			IF curStep = 1 THEN
				IF ZeitPuls > loc_ET_ms THEN
					RestzeitPuls := ZeitPuls - loc_ET_ms;
				ELSE
					RestzeitPuls := 0;
				END_IF;
				RestzeitPause := ZeitPause;
			ELSE
				RestzeitPuls := ZeitPuls;
				IF ZeitPause > loc_ET_ms THEN
					RestzeitPause := ZeitPause - loc_ET_ms;
				ELSE
					RestzeitPause := 0;
				END_IF;
			END_IF;
		END_IF;

	END_IF;

ELSE
	(* keine Freigabe -> Schrittkette ruecksetzen *)
	PulsOut       := FALSE;
	PauseOut      := FALSE;
	RestzeitPuls  := 0;
	RestzeitPause := 0;
	TON_PulsPause(IN := FALSE, PT := 0);
	curStep       := 0;
	stateEntry    := TRUE;
END_IF;
END_FUNCTION_BLOCK

FUNCTION_BLOCK fbRestzeit
  VAR
    i : INT;
    ii : INT;
    stundeEndeTag : INT;
    minRestTag : UINT;
    minRestFolgetag : UINT;
    minRestGesamt : UINT;
    restStd : UINT;
  END_VAR
  VAR_INPUT
    Freigabe : BOOL;
    AktuelleStunde : USINT;  (* 0..23 *)
    AktuelleMinute : USINT;  (* 0..59 *)
  END_VAR
  VAR_OUTPUT
    ZeitfensterAktiv : BOOL;
    RestzeitStundenOut : UINT;
    RestzeitMinutenOut : UINT;
  END_VAR
  VAR_IN_OUT
    ZeitfensterIn : ARRAY[0..23] OF BOOL;
  END_VAR

IF Freigabe THEN
    ZeitfensterAktiv := ZeitfensterIn[AktuelleStunde];

    (* Ende des aktuellen (gleichbleibenden) Blocks heute suchen *)
    stundeEndeTag := 23;
    FOR i := TO_INT(AktuelleStunde) + 1 TO 23 DO
        IF ZeitfensterIn[i] <> ZeitfensterAktiv THEN
            stundeEndeTag := i - 1;
            EXIT;
        END_IF;
    END_FOR;

    (* Restminuten heute *)
    minRestTag := 60 - AktuelleMinute;
    IF stundeEndeTag > TO_INT(AktuelleStunde) THEN
        minRestTag := minRestTag + TO_UINT(stundeEndeTag - TO_INT(AktuelleStunde)) * 60;
    END_IF;

    (* Folgetag nur, wenn Block bis 23 Uhr durchlaeuft *)
    minRestFolgetag := 0;
    IF stundeEndeTag = 23 THEN
        FOR ii := 0 TO 23 DO
            IF ZeitfensterIn[ii] = ZeitfensterAktiv THEN
                minRestFolgetag := minRestFolgetag + 60;
            ELSE
                EXIT;
            END_IF;
        END_FOR;
    END_IF;

    minRestGesamt := minRestTag + minRestFolgetag;
    restStd := minRestGesamt / 60;
    IF restStd <= 24 THEN
        RestzeitStundenOut := restStd;
        RestzeitMinutenOut := minRestGesamt - (restStd * 60);
    ELSE
        RestzeitStundenOut := 65535;   (* >24h -> keine Anzeige *)
        RestzeitMinutenOut := 65535;
    END_IF;
ELSE
    ZeitfensterAktiv   := FALSE;
    RestzeitStundenOut := 65535;
    RestzeitMinutenOut := 65535;
END_IF;
END_FUNCTION_BLOCK

FUNCTION_BLOCK fbBetriebsstunden
  VAR
    Sekunden : USINT;
  END_VAR
  VAR_INPUT
    Aktiv : BOOL;
    sekTick : BOOL;  (* 1-Sekunden-Puls *)
    Reset : BOOL;
  END_VAR
  VAR_IN_OUT
    Minuten : UINT;  (* Retain-Global, 0..59 *)
    Stunden : UDINT;  (* Retain-Global *)
  END_VAR

IF Reset THEN
    Sekunden := 0;  Minuten := 0;  Stunden := 0;
ELSIF (Aktiv AND sekTick) THEN
    IF Sekunden < 59 THEN
        Sekunden := Sekunden + 1;
    ELSE
        Sekunden := 0;
        IF Minuten < 59 THEN
            Minuten := Minuten + 1;
        ELSE
            Minuten := 0;
            Stunden := Stunden + 1;
        END_IF;
    END_IF;
END_IF;
END_FUNCTION_BLOCK

FUNCTION fcSetBitInBitmask : UDINT
  VAR
    ValBit : UDINT;
  END_VAR
  VAR_INPUT
    Bitmask : UDINT;
    BitNr : USINT;
  END_VAR

// Bitstelle in Wert umwandeln
ValBit := SHL(UDINT#1, BitNr);

// Bit in Bitmaske setzen
fcSetBitInBitmask := Bitmask OR ValBit;
END_FUNCTION

FUNCTION fcClearBitInBitmask : UDINT
  VAR
    ValBit : UDINT;
  END_VAR
  VAR_INPUT
    Bitmask : UDINT;
    BitNr : USINT;
  END_VAR

// Bitstelle in Wert umwandeln
ValBit := SHL(UDINT#1, BitNr);

// Bit in Bitmaske löschen
fcClearBitInBitmask := Bitmask AND NOT ValBit;
END_FUNCTION

FUNCTION fcResetBitmask : UDINT

fcResetBitmask := TO_UDINT(0);
END_FUNCTION

CONFIGURATION Configuration
  RESOURCE Resource ON PLC
    VAR_GLOBAL  (* var_glob *)
      gAktModus : eBetriebsmodus := BETRIEB;
      gStatusAnlage : T_StatAnlage;
      gBetriebsparameter : T_Betriebsparameter;
      gAktoren : T_Aktor;
      gIoTest : T_IoTest;
      gCmdAnlage : T_CmdAnlage;
      Strombegrenzung : fbTrockStrombegr;  (* Strombegrenzung Logik *)
      gQuitErr : BOOL;  (* Fehler quittieren *)
      IBN_FALSE : BOOL;  (* Inbetriebnahmemerker false *)
      IBN_TRUE : BOOL;  (* Inbetriebnahmemerker true *)
      diBox1Offen : BOOL;  (* Rückmeldung Box 1 offen *)
      diBox1Geschl : BOOL;  (* Rückmeldung Box 1 geschlossen *)
      diBox2Offen : BOOL;  (* Rückmeldung Box 2 offen *)
      diBox2Geschl : BOOL;  (* Rückmeldung Box 2 geschlossen *)
      diBetriebLuftaufber : BOOL;  (* Betriebsmeldung Luftaufbereitung *)
      diBetriebVentilator : BOOL;  (* Betriebsmeldung Ventilator *)
      aiFrischluftTemp : REAL;  (* Frischlufttemperatur *)
      aiFrischluftFeucht : REAL;  (* Frischluftfeuchte *)
      aiAbluftBox1Temp : REAL;  (* Ablufttemperatur Box 1 *)
      aiAbluftBox1Feucht : REAL;  (* Abluftfeuchte Box 1 *)
      aiTrockenluftTemp : REAL;  (* Trockenlufttemperatur *)
      aiTrockenluftFeucht : REAL;  (* Trockenluftfeuchte *)
      aiAbluftBox2Temp : REAL;  (* Ablufttemperatur Box 2 *)
      aiAbluftBox2Feucht : REAL;  (* Abluftfeuchte Box 2 *)
      aiStocktemp : REAL;  (* Stock- bzw. Produkttemperatur *)
      doFrgLuftaufber : BOOL;  (* Freigabe Luftaufbereiter (Digitaler Ausgang) *)
      doFrgBox1 : BOOL;  (* Freigabe Box 1 (z.B. Klappe / Aktor Box 1) *)
      doFrgBox2 : BOOL;  (* Freigabe Box 2 (z.B. Klappe / Aktor Box 2) *)
      doFrgAbluftventilator : BOOL;  (* Freigabe Abluftventilator *)
      doFrgVentilator : BOOL;  (* Freigabe Ventilator *)
      aoFuVentilator : REAL;  (* Sollwert Frequenzumrichter Ventilator [%] *)
      aoLeistVorgLuftaufber : REAL;  (* Leistungsvorgabe Luftaufbereiter [%] *)
      gudTemp : UDINT;
    END_VAR
    VAR_GLOBAL CONSTANT  (* var_glob_$Constant *)
      gPlcSwVersion : STRING := 'v1.0.0';  (* PLC Software Version *)
      gPlcKonfigId : UINT := 8;  (* PLC Konfiguration [8...2.04] *)
    END_VAR
    VAR_GLOBAL  (* varAlarm *)
      gAlarmBetriebLuftaufber : BOOL;
      gAlarmBetriebVentilator : BOOL;
    END_VAR
    VAR_GLOBAL  (* var_VisuIo *)
      hmiNutzungsdaten : ST_HmiNutzungsdaten;
    END_VAR
    VAR_GLOBAL RETAIN  (* var_glob_retain *)
      gBstBox1Min : UINT;
      gBstBox1Std : UDINT;
      gBstBox2Min : UINT;
      gBstBox2Std : UDINT;
    END_VAR
  END_RESOURCE
END_CONFIGURATION
